Staubli VAL3: encoder.pgx

program encoder()
  local bool l_bRisenEdge
  local num l_nTriggerCount
begin
  // This routine manages the encoder input of the Wago Module 750-631
  //
  //
  //----------------------------------------------------------------
  //
  l_nTriggerCount=0
  do
    // Read current encoder position
    nEncValue=aioGet(aiEncCurrentPos)
    //
    // Re-enable the latch feature
    if (bLatchEnabled==true) and (diEncLatched==false)
      doEnableLatch=true
    endIf
    //
    // Check if latch feature is enabled by conveyor library
    if bLatchEnabled==true
      // check for rising edge on the Latch Input
      call _DetectIOEdge((diEncLatched==true),bMemoLatchState,l_bRisenEdge)
      //
      if l_bRisenEdge==true
        // Check number of latch for part detection
        l_nTriggerCount=l_nTriggerCount+1
        if l_nTriggerCount>=nLatchPeriod
          // Compute Latched value
          nEncLatchedVal=aioGet(aiEncLatchedPos)
          bPartLatched=true
          l_nTriggerCount=0
        endIf
        doEnableLatch=false
      endIf
    endIf
    //
    delay(0)
  until false
end
